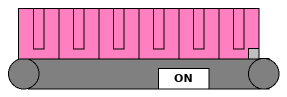
embedded screen at (210,0)-(251,51): VC_Part
embedded screen at (240,40)-(251,51): VC_sensor
embedded screen at (170,0)-(211,51): VC_Part
embedded screen at (130,0)-(171,51): VC_Part
embedded screen at (90,0)-(131,51): VC_Part
embedded screen at (50,0)-(91,51): VC_Part
embedded screen at (10,0)-(51,51): VC_Part
rectangle at (150,60)-(201,81): text "OFF"
rectangle at (150,60)-(201,81): text "ON"; invisible if NOT $MotOn$
3 more shapes without text or variables
*)

(* Visualisation Simulator/MachineComponents/VC_Simu_Drill
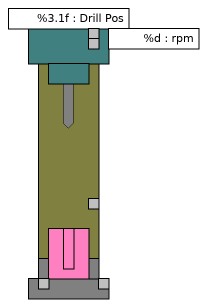
rectangle at (20,20)-(101,56): y offset $FB$.fBasePos_Y
rectangle at (0,0)-(121,21): text "%3.1f : Drill Pos"; shows $FB$.fLift_CurrentPos
embedded screen at (80,20)-(91,31): VC_sensor
embedded screen at (80,190)-(91,201): VC_sensor
embedded screen at (80,30)-(91,41): VC_sensor
polygon at (55,75)-(65,120): alarm colour if $FB$.iRPMCurrent > 0; y offset $FB$.fBasePos_Y
rectangle at (40,55)-(81,76): y offset $FB$.fBasePos_Y
rectangle at (30,250)-(41,271): x offset - $FB$.fPosJawDiff
rectangle at (80,250)-(91,271): x offset $FB$.fPosJawDiff
embedded screen at (40,220)-(81,271): VC_Part
embedded screen at (90,270)-(101,281): VC_sensor
embedded screen at (30,270)-(41,281): VC_sensor
rectangle at (100,20)-(191,41): text "%d : rpm"; shows $FB$.iRPMCurrent
2 more shapes without text or variables
*)

(* Visualisation Simulator/MachineComponents/VC_Simu_Manipulator
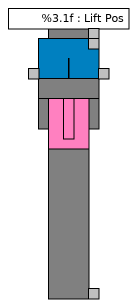
rectangle at (70,40)-(131,81): y offset $FB$.fBasePos_Y
rectangle at (100,60)-(101,81): left $FB$.fPos_Beam_L; right $FB$.fPos_Beam_R; y offset $FB$.fBasePos_Y
rectangle at (70,80)-(131,101): x offset $FB$.fPos_X; y offset $FB$.fBasePos_Y
rectangle at (70,100)-(81,131): x offset $FB$.fPos_X - $FB$.fPosFingerDiff; y offset $FB$.fBasePos_Y
rectangle at (120,100)-(131,131): x offset $FB$.fPos_X + $FB$.fPosFingerDiff; y offset $FB$.fBasePos_Y
embedded screen at (80,100)-(121,151): VC_Part
rectangle at (40,10)-(161,31): text "%3.1f : Lift Pos"; shows $FB$.fLift_CurrentPos
embedded screen at (120,30)-(131,41): VC_sensor
embedded screen at (120,290)-(131,301): VC_sensor
embedded screen at (120,40)-(131,51): VC_sensor
embedded screen at (130,70)-(141,81): VC_sensor
embedded screen at (60,70)-(71,81): VC_sensor
1 more shapes without text or variables
*)

(* Visualisation Simulator/MachineComponents/VC_SimuMach_Controls
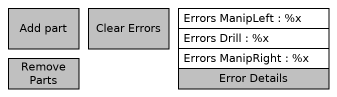
rounded rectangle at (0,0)-(71,41): text "Add part"; alarm colour if PRG_Simulator.bAddPartOnConvIn; taps PRG_Simulator.bAddPartOnConvIn
rounded rectangle at (80,0)-(161,41): text "Clear Errors"; alarm colour if PRG_Simulator.bClearErrors; taps PRG_Simulator.bClearErrors
rectangle at (170,0)-(321,21): text "Errors ManipLeft : %x"; shows PRG_Simulator.wError_ManipL; alarm colour if PRG_Simulator.wError_ManipL > 0
rounded rectangle at (0,50)-(71,81): text "Remove / Parts"; alarm colour if PRG_Simulator.bClearSystem; taps PRG_Simulator.bClearSystem
rectangle at (170,20)-(321,41): text "Errors Drill : %x"; shows PRG_Simulator.wError_Drill; alarm colour if PRG_Simulator.wError_Drill > 0
rectangle at (170,40)-(321,61): text "Errors ManipRight : %x"; shows PRG_Simulator.wError_ManipR; alarm colour if PRG_Simulator.wError_ManipR > 0
rounded rectangle at (170,60)-(321,81): text "Error Details"; opens VC_ErrorDetails
*)

(* Visualisation Simulator/VISU_SimulatedMachine
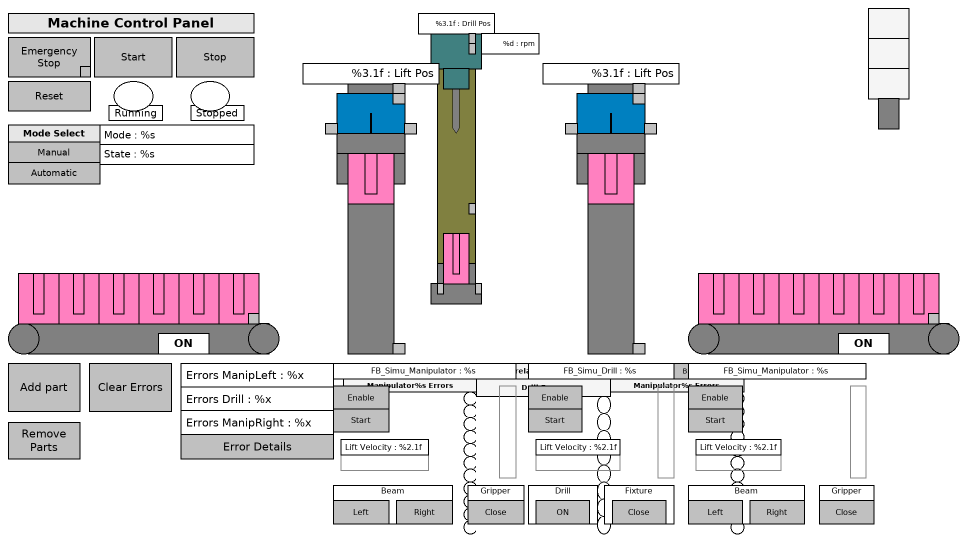
embedded screen at (335,320)-(736,491): VC_ErrorDetails
embedded screen at (0,-30)-(246,141): VC_Panel_MachineControl
embedded screen at (410,-30)-(531,261): VC_Simu_Drill
embedded screen at (0,230)-(271,311): VC_Simu_Conv_In
embedded screen at (0,320)-(326,416): VC_SimuMach_Controls
embedded screen at (325,320)-(516,481): VC_FB_Simu_Manipulator
embedded screen at (250,10)-(431,311): VC_Simu_Manipulator
embedded screen at (490,10)-(671,311): VC_Simu_Manipulator
embedded screen at (680,320)-(866,481): VC_FB_Simu_Manipulator
embedded screen at (520,320)-(666,481): VC_FB_Simu_Drill
embedded screen at (680,230)-(951,311): VC_Simu_Conv_In
embedded screen at (860,-35)-(901,86): VC_Beacon
*)
